// TIA Portal V16 export
// export: Created 2022-11-17T15:49:30.6302433Z, ExportSetting WithDefaults, DisplayName Totally Integrated Automation Portal, DisplayVersion V16 Update 6, DisplayName TIA Portal Version Control Interface, DisplayVersion V16 Update 2, DisplayName TIA Portal Openness, DisplayVersion V16 Update 6, DisplayName SINAMICS Startdrive Advanced, DisplayVersion V16 Update 5, DisplayName SINAMICS Startdrive G130, G150, S120, S150, SINAMICS MV, S210, DisplayVersion V16 Update 5, DisplayName SINAMICS Startdrive G110M, G120, G120C, G120D, G120P, G115D, DisplayVersion V16 Update 5, DisplayName STEP 7 Professional, DisplayVersion V16 Update 6, DisplayName STEP 7 Safety, DisplayVersion V16, DisplayName WinCC Advanced, DisplayVersion V16 Update 6
FUNCTION "FC90_PageManagement" : Void   // FC90, LAD
{ S7_Optimized_Access := 'FALSE' }
VERSION : 0.1
// stored: AutoNumber false, IsIECCheckEnabled false, SetENOAutomatically false, UDAEnableTagReadback false
   VAR_TEMP
      CurrentPage : Int;
      PageBkwRequest : Int;
      PageFwRequest : Int;
   END_VAR
   VAR_TEMP   // added for the SCL form of the ladder/FBD networks
      _w1 : Bool;
   END_VAR
BEGIN

REGION Network 1
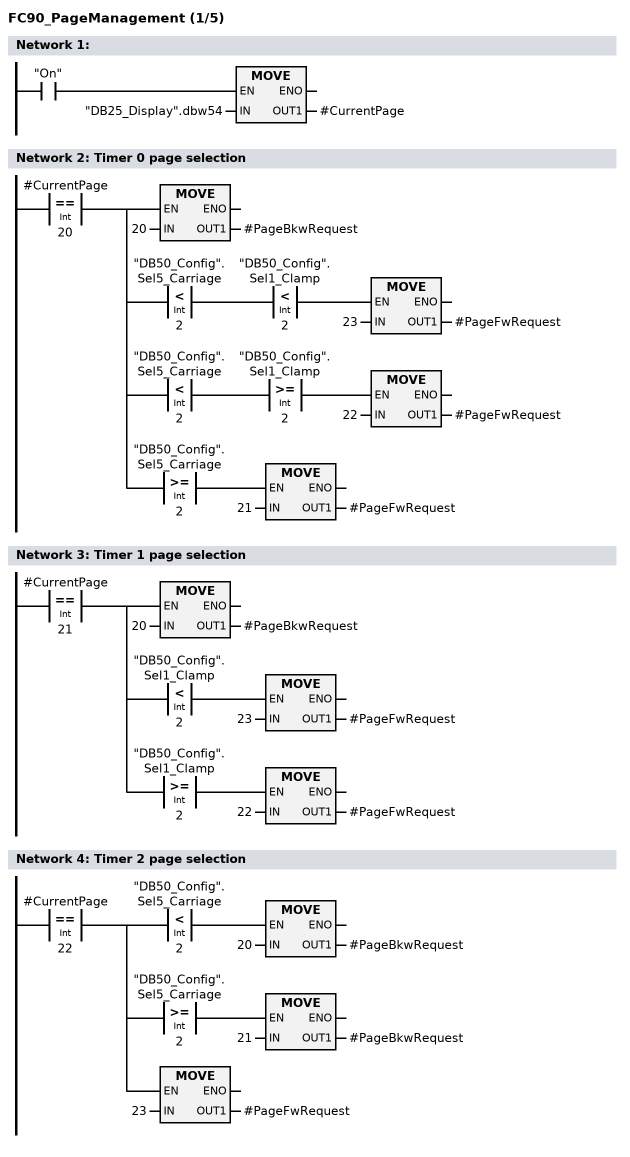
   RUNG wire#powerrail
      Contact( "On" )
      { S7_GenerateENO := "TRUE" } Move(in := "DB25_Display".dbw54, out1 => #CurrentPage)
   END_RUNG
   // the same network as SCL:
   IF "On" THEN #CurrentPage := "DB25_Display".dbw54; END_IF;
END_REGION

REGION Network 2: Timer 0 page selection
   RUNG wire#powerrail
      { S7_Templates := "SrcType := Int" } EQ_Contact(in1 := #CurrentPage, in2 := 20)
      wire#w1
      { S7_GenerateENO := "TRUE" } Move(in := 20, out1 => #PageBkwRequest)
   END_RUNG
   RUNG wire#w1
      { S7_Templates := "SrcType := Int" } LT_Contact(in1 := "DB50_Config".Sel5_Carriage, in2 := 2)
      { S7_Templates := "SrcType := Int" } LT_Contact(in1 := "DB50_Config".Sel1_Clamp, in2 := 2)
      { S7_GenerateENO := "TRUE" } Move(in := 23, out1 => #PageFwRequest)
   END_RUNG
   RUNG wire#w1
      { S7_Templates := "SrcType := Int" } LT_Contact(in1 := "DB50_Config".Sel5_Carriage, in2 := 2)
      { S7_Templates := "SrcType := Int" } GE_Contact(in1 := "DB50_Config".Sel1_Clamp, in2 := 2)
      { S7_GenerateENO := "TRUE" } Move(in := 22, out1 => #PageFwRequest)
   END_RUNG
   RUNG wire#w1
      { S7_Templates := "SrcType := Int" } GE_Contact(in1 := "DB50_Config".Sel5_Carriage, in2 := 2)
      { S7_GenerateENO := "TRUE" } Move(in := 21, out1 => #PageFwRequest)
   END_RUNG
   // the same network as SCL:
   #_w1 := #CurrentPage = 20;
   IF #_w1 THEN #PageBkwRequest := 20; END_IF;
   IF #_w1 AND ("DB50_Config".Sel5_Carriage < 2) AND ("DB50_Config".Sel1_Clamp < 2) THEN
       #PageFwRequest := 23;
   END_IF;
   IF #_w1 AND ("DB50_Config".Sel5_Carriage < 2) AND ("DB50_Config".Sel1_Clamp >= 2) THEN
       #PageFwRequest := 22;
   END_IF;
   IF #_w1 AND ("DB50_Config".Sel5_Carriage >= 2) THEN #PageFwRequest := 21; END_IF;
END_REGION

REGION Network 3: Timer 1 page selection
   RUNG wire#powerrail
      { S7_Templates := "SrcType := Int" } EQ_Contact(in1 := #CurrentPage, in2 := 21)
      wire#w1
      { S7_GenerateENO := "TRUE" } Move(in := 20, out1 => #PageBkwRequest)
   END_RUNG
   RUNG wire#w1
      { S7_Templates := "SrcType := Int" } LT_Contact(in1 := "DB50_Config".Sel1_Clamp, in2 := 2)
      { S7_GenerateENO := "TRUE" } Move(in := 23, out1 => #PageFwRequest)
   END_RUNG
   RUNG wire#w1
      { S7_Templates := "SrcType := Int" } GE_Contact(in1 := "DB50_Config".Sel1_Clamp, in2 := 2)
      { S7_GenerateENO := "TRUE" } Move(in := 22, out1 => #PageFwRequest)
   END_RUNG
   // the same network as SCL:
   #_w1 := #CurrentPage = 21;
   IF #_w1 THEN #PageBkwRequest := 20; END_IF;
   IF #_w1 AND ("DB50_Config".Sel1_Clamp < 2) THEN #PageFwRequest := 23; END_IF;
   IF #_w1 AND ("DB50_Config".Sel1_Clamp >= 2) THEN #PageFwRequest := 22; END_IF;
END_REGION

REGION Network 4: Timer 2 page selection
   RUNG wire#powerrail
      { S7_Templates := "SrcType := Int" } EQ_Contact(in1 := #CurrentPage, in2 := 22)
      wire#w1
      { S7_Templates := "SrcType := Int" } LT_Contact(in1 := "DB50_Config".Sel5_Carriage, in2 := 2)
      { S7_GenerateENO := "TRUE" } Move(in := 20, out1 => #PageBkwRequest)
   END_RUNG
   RUNG wire#w1
      { S7_Templates := "SrcType := Int" } GE_Contact(in1 := "DB50_Config".Sel5_Carriage, in2 := 2)
      { S7_GenerateENO := "TRUE" } Move(in := 21, out1 => #PageBkwRequest)
   END_RUNG
   RUNG wire#w1
      { S7_GenerateENO := "TRUE" } Move(in := 23, out1 => #PageFwRequest)
   END_RUNG
   // the same network as SCL:
   #_w1 := #CurrentPage = 22;
   IF #_w1 AND ("DB50_Config".Sel5_Carriage < 2) THEN #PageBkwRequest := 20; END_IF;
   IF #_w1 AND ("DB50_Config".Sel5_Carriage >= 2) THEN #PageBkwRequest := 21; END_IF;
   IF #_w1 THEN #PageFwRequest := 23; END_IF;
END_REGION

REGION Network 5: Timer 3 page selection
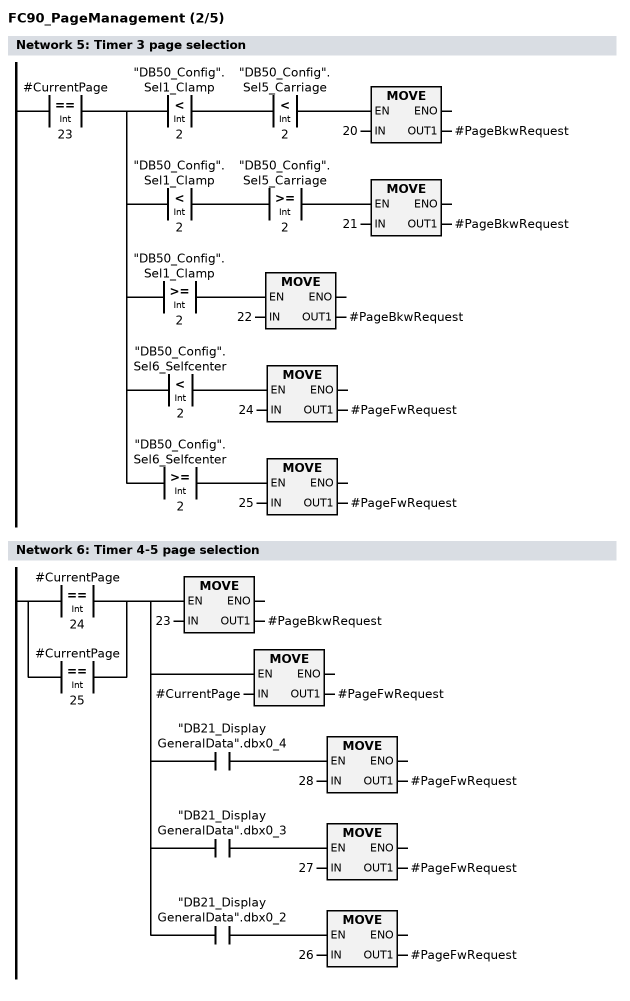
   RUNG wire#powerrail
      { S7_Templates := "SrcType := Int" } EQ_Contact(in1 := #CurrentPage, in2 := 23)
      wire#w1
      { S7_Templates := "SrcType := Int" } LT_Contact(in1 := "DB50_Config".Sel1_Clamp, in2 := 2)
      { S7_Templates := "SrcType := Int" } LT_Contact(in1 := "DB50_Config".Sel5_Carriage, in2 := 2)
      { S7_GenerateENO := "TRUE" } Move(in := 20, out1 => #PageBkwRequest)
   END_RUNG
   RUNG wire#w1
      { S7_Templates := "SrcType := Int" } LT_Contact(in1 := "DB50_Config".Sel1_Clamp, in2 := 2)
      { S7_Templates := "SrcType := Int" } GE_Contact(in1 := "DB50_Config".Sel5_Carriage, in2 := 2)
      { S7_GenerateENO := "TRUE" } Move(in := 21, out1 => #PageBkwRequest)
   END_RUNG
   RUNG wire#w1
      { S7_Templates := "SrcType := Int" } GE_Contact(in1 := "DB50_Config".Sel1_Clamp, in2 := 2)
      { S7_GenerateENO := "TRUE" } Move(in := 22, out1 => #PageBkwRequest)
   END_RUNG
   RUNG wire#w1
      { S7_Templates := "SrcType := Int" } LT_Contact(in1 := "DB50_Config".Sel6_Selfcenter, in2 := 2)
      { S7_GenerateENO := "TRUE" } Move(in := 24, out1 => #PageFwRequest)
   END_RUNG
   RUNG wire#w1
      { S7_Templates := "SrcType := Int" } GE_Contact(in1 := "DB50_Config".Sel6_Selfcenter, in2 := 2)
      { S7_GenerateENO := "TRUE" } Move(in := 25, out1 => #PageFwRequest)
   END_RUNG
   // the same network as SCL:
   #_w1 := #CurrentPage = 23;
   IF #_w1 AND ("DB50_Config".Sel1_Clamp < 2) AND ("DB50_Config".Sel5_Carriage < 2) THEN
       #PageBkwRequest := 20;
   END_IF;
   IF #_w1 AND ("DB50_Config".Sel1_Clamp < 2) AND ("DB50_Config".Sel5_Carriage >= 2) THEN
       #PageBkwRequest := 21;
   END_IF;
   IF #_w1 AND ("DB50_Config".Sel1_Clamp >= 2) THEN #PageBkwRequest := 22; END_IF;
   IF #_w1 AND ("DB50_Config".Sel6_Selfcenter < 2) THEN #PageFwRequest := 24; END_IF;
   IF #_w1 AND ("DB50_Config".Sel6_Selfcenter >= 2) THEN #PageFwRequest := 25; END_IF;
END_REGION

REGION Network 6: Timer 4-5 page selection
   RUNG wire#powerrail
      { S7_Templates := "SrcType := Int" } EQ_Contact(in1 := #CurrentPage, in2 := 24)
      wire#w1
      { S7_GenerateENO := "TRUE" } Move(in := 23, out1 => #PageBkwRequest)
   END_RUNG
   RUNG wire#powerrail
      { S7_Templates := "SrcType := Int" } EQ_Contact(in1 := #CurrentPage, in2 := 25)
   END_RUNG wire#w1
   RUNG wire#w1
      { S7_GenerateENO := "TRUE" } Move(in := #CurrentPage, out1 => #PageFwRequest)
   END_RUNG
   RUNG wire#w1
      Contact( "DB21_DisplayGeneralData".dbx0_4 )
      { S7_GenerateENO := "TRUE" } Move(in := 28, out1 => #PageFwRequest)
   END_RUNG
   RUNG wire#w1
      Contact( "DB21_DisplayGeneralData".dbx0_3 )
      { S7_GenerateENO := "TRUE" } Move(in := 27, out1 => #PageFwRequest)
   END_RUNG
   RUNG wire#w1
      Contact( "DB21_DisplayGeneralData".dbx0_2 )
      { S7_GenerateENO := "TRUE" } Move(in := 26, out1 => #PageFwRequest)
   END_RUNG
   // the same network as SCL:
   #_w1 := (#CurrentPage = 24) OR (#CurrentPage = 25);
   IF #_w1 THEN
       #PageBkwRequest := 23;
       #PageFwRequest := #CurrentPage;
   END_IF;
   IF #_w1 AND "DB21_DisplayGeneralData".dbx0_4 THEN #PageFwRequest := 28; END_IF;
   IF #_w1 AND "DB21_DisplayGeneralData".dbx0_3 THEN #PageFwRequest := 27; END_IF;
   IF #_w1 AND "DB21_DisplayGeneralData".dbx0_2 THEN #PageFwRequest := 26; END_IF;
END_REGION

REGION Network 7: Timer 6 page selection
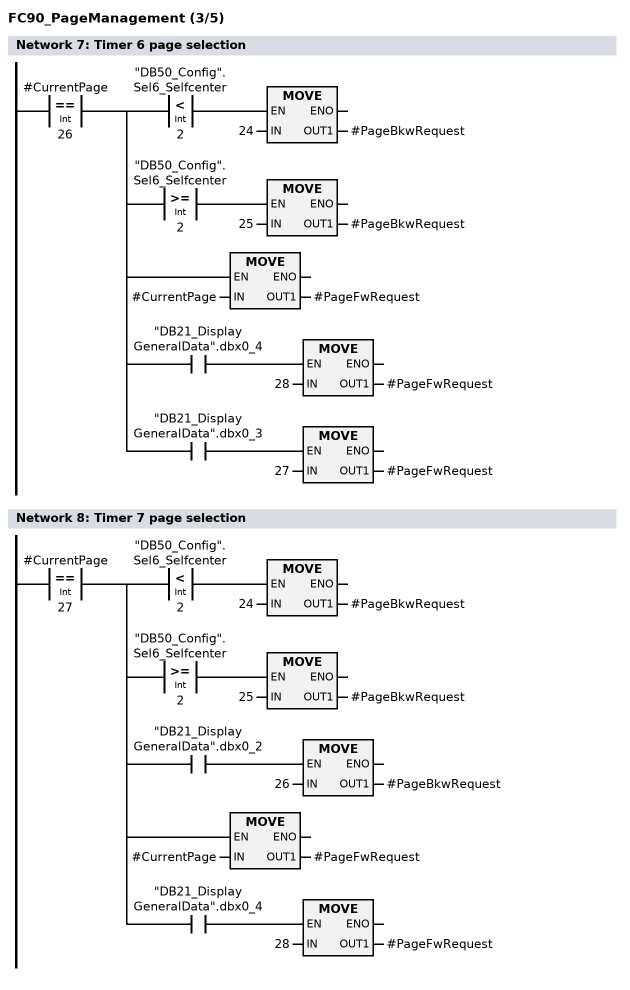
   RUNG wire#powerrail
      { S7_Templates := "SrcType := Int" } EQ_Contact(in1 := #CurrentPage, in2 := 26)
      wire#w1
      { S7_Templates := "SrcType := Int" } LT_Contact(in1 := "DB50_Config".Sel6_Selfcenter, in2 := 2)
      { S7_GenerateENO := "TRUE" } Move(in := 24, out1 => #PageBkwRequest)
   END_RUNG
   RUNG wire#w1
      { S7_Templates := "SrcType := Int" } GE_Contact(in1 := "DB50_Config".Sel6_Selfcenter, in2 := 2)
      { S7_GenerateENO := "TRUE" } Move(in := 25, out1 => #PageBkwRequest)
   END_RUNG
   RUNG wire#w1
      { S7_GenerateENO := "TRUE" } Move(in := #CurrentPage, out1 => #PageFwRequest)
   END_RUNG
   RUNG wire#w1
      Contact( "DB21_DisplayGeneralData".dbx0_4 )
      { S7_GenerateENO := "TRUE" } Move(in := 28, out1 => #PageFwRequest)
   END_RUNG
   RUNG wire#w1
      Contact( "DB21_DisplayGeneralData".dbx0_3 )
      { S7_GenerateENO := "TRUE" } Move(in := 27, out1 => #PageFwRequest)
   END_RUNG
   // the same network as SCL:
   #_w1 := #CurrentPage = 26;
   IF #_w1 AND ("DB50_Config".Sel6_Selfcenter < 2) THEN #PageBkwRequest := 24; END_IF;
   IF #_w1 AND ("DB50_Config".Sel6_Selfcenter >= 2) THEN #PageBkwRequest := 25; END_IF;
   IF #_w1 THEN #PageFwRequest := #CurrentPage; END_IF;
   IF #_w1 AND "DB21_DisplayGeneralData".dbx0_4 THEN #PageFwRequest := 28; END_IF;
   IF #_w1 AND "DB21_DisplayGeneralData".dbx0_3 THEN #PageFwRequest := 27; END_IF;
END_REGION

REGION Network 8: Timer 7 page selection
   RUNG wire#powerrail
      { S7_Templates := "SrcType := Int" } EQ_Contact(in1 := #CurrentPage, in2 := 27)
      wire#w1
      { S7_Templates := "SrcType := Int" } LT_Contact(in1 := "DB50_Config".Sel6_Selfcenter, in2 := 2)
      { S7_GenerateENO := "TRUE" } Move(in := 24, out1 => #PageBkwRequest)
   END_RUNG
   RUNG wire#w1
      { S7_Templates := "SrcType := Int" } GE_Contact(in1 := "DB50_Config".Sel6_Selfcenter, in2 := 2)
      { S7_GenerateENO := "TRUE" } Move(in := 25, out1 => #PageBkwRequest)
   END_RUNG
   RUNG wire#w1
      Contact( "DB21_DisplayGeneralData".dbx0_2 )
      { S7_GenerateENO := "TRUE" } Move(in := 26, out1 => #PageBkwRequest)
   END_RUNG
   RUNG wire#w1
      { S7_GenerateENO := "TRUE" } Move(in := #CurrentPage, out1 => #PageFwRequest)
   END_RUNG
   RUNG wire#w1
      Contact( "DB21_DisplayGeneralData".dbx0_4 )
      { S7_GenerateENO := "TRUE" } Move(in := 28, out1 => #PageFwRequest)
   END_RUNG
   // the same network as SCL:
   #_w1 := #CurrentPage = 27;
   IF #_w1 AND ("DB50_Config".Sel6_Selfcenter < 2) THEN #PageBkwRequest := 24; END_IF;
   IF #_w1 AND ("DB50_Config".Sel6_Selfcenter >= 2) THEN #PageBkwRequest := 25; END_IF;
   IF #_w1 AND "DB21_DisplayGeneralData".dbx0_2 THEN #PageBkwRequest := 26; END_IF;
   IF #_w1 THEN #PageFwRequest := #CurrentPage; END_IF;
   IF #_w1 AND "DB21_DisplayGeneralData".dbx0_4 THEN #PageFwRequest := 28; END_IF;
END_REGION

REGION Network 9: Timer 8 page selection
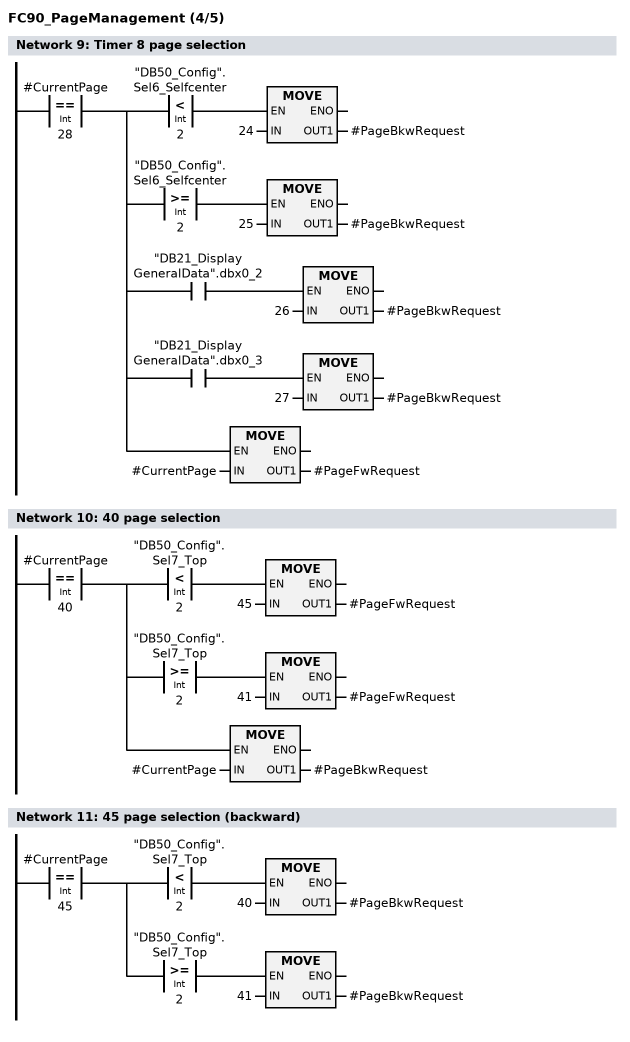
   RUNG wire#powerrail
      { S7_Templates := "SrcType := Int" } EQ_Contact(in1 := #CurrentPage, in2 := 28)
      wire#w1
      { S7_Templates := "SrcType := Int" } LT_Contact(in1 := "DB50_Config".Sel6_Selfcenter, in2 := 2)
      { S7_GenerateENO := "TRUE" } Move(in := 24, out1 => #PageBkwRequest)
   END_RUNG
   RUNG wire#w1
      { S7_Templates := "SrcType := Int" } GE_Contact(in1 := "DB50_Config".Sel6_Selfcenter, in2 := 2)
      { S7_GenerateENO := "TRUE" } Move(in := 25, out1 => #PageBkwRequest)
   END_RUNG
   RUNG wire#w1
      Contact( "DB21_DisplayGeneralData".dbx0_2 )
      { S7_GenerateENO := "TRUE" } Move(in := 26, out1 => #PageBkwRequest)
   END_RUNG
   RUNG wire#w1
      Contact( "DB21_DisplayGeneralData".dbx0_3 )
      { S7_GenerateENO := "TRUE" } Move(in := 27, out1 => #PageBkwRequest)
   END_RUNG
   RUNG wire#w1
      { S7_GenerateENO := "TRUE" } Move(in := #CurrentPage, out1 => #PageFwRequest)
   END_RUNG
   // the same network as SCL:
   #_w1 := #CurrentPage = 28;
   IF #_w1 AND ("DB50_Config".Sel6_Selfcenter < 2) THEN #PageBkwRequest := 24; END_IF;
   IF #_w1 AND ("DB50_Config".Sel6_Selfcenter >= 2) THEN #PageBkwRequest := 25; END_IF;
   IF #_w1 AND "DB21_DisplayGeneralData".dbx0_2 THEN #PageBkwRequest := 26; END_IF;
   IF #_w1 AND "DB21_DisplayGeneralData".dbx0_3 THEN #PageBkwRequest := 27; END_IF;
   IF #_w1 THEN #PageFwRequest := #CurrentPage; END_IF;
END_REGION

REGION Network 10: 40 page selection
   RUNG wire#powerrail
      { S7_Templates := "SrcType := Int" } EQ_Contact(in1 := #CurrentPage, in2 := 40)
      wire#w1
      { S7_Templates := "SrcType := Int" } LT_Contact(in1 := "DB50_Config".Sel7_Top, in2 := 2)
      { S7_GenerateENO := "TRUE" } Move(in := 45, out1 => #PageFwRequest)
   END_RUNG
   RUNG wire#w1
      { S7_Templates := "SrcType := Int" } GE_Contact(in1 := "DB50_Config".Sel7_Top, in2 := 2)
      { S7_GenerateENO := "TRUE" } Move(in := 41, out1 => #PageFwRequest)
   END_RUNG
   RUNG wire#w1
      { S7_GenerateENO := "TRUE" } Move(in := #CurrentPage, out1 => #PageBkwRequest)
   END_RUNG
   // the same network as SCL:
   #_w1 := #CurrentPage = 40;
   IF #_w1 AND ("DB50_Config".Sel7_Top < 2) THEN #PageFwRequest := 45; END_IF;
   IF #_w1 AND ("DB50_Config".Sel7_Top >= 2) THEN #PageFwRequest := 41; END_IF;
   IF #_w1 THEN #PageBkwRequest := #CurrentPage; END_IF;
END_REGION

REGION Network 11: 45 page selection (backward)
   RUNG wire#powerrail
      { S7_Templates := "SrcType := Int" } EQ_Contact(in1 := #CurrentPage, in2 := 45)
      wire#w1
      { S7_Templates := "SrcType := Int" } LT_Contact(in1 := "DB50_Config".Sel7_Top, in2 := 2)
      { S7_GenerateENO := "TRUE" } Move(in := 40, out1 => #PageBkwRequest)
   END_RUNG
   RUNG wire#w1
      { S7_Templates := "SrcType := Int" } GE_Contact(in1 := "DB50_Config".Sel7_Top, in2 := 2)
      { S7_GenerateENO := "TRUE" } Move(in := 41, out1 => #PageBkwRequest)
   END_RUNG
   // the same network as SCL:
   #_w1 := #CurrentPage = 45;
   IF #_w1 AND ("DB50_Config".Sel7_Top < 2) THEN #PageBkwRequest := 40; END_IF;
   IF #_w1 AND ("DB50_Config".Sel7_Top >= 2) THEN #PageBkwRequest := 41; END_IF;
END_REGION

REGION Network 12
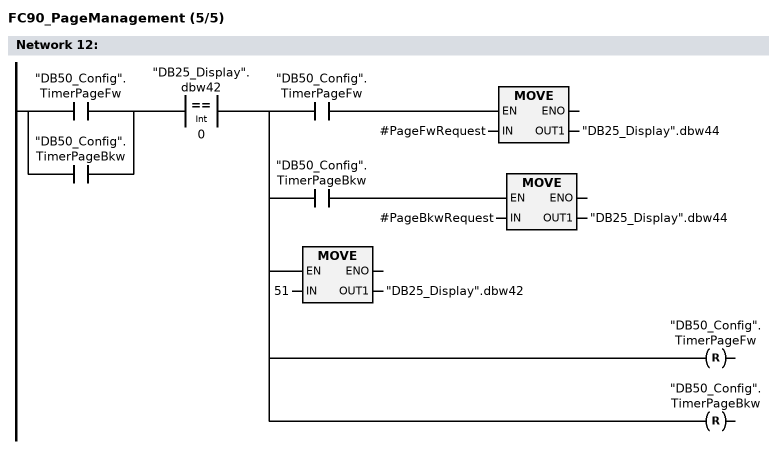
   RUNG wire#powerrail
      Contact( "DB50_Config".TimerPageFw )
      wire#w1
      { S7_Templates := "SrcType := Int" } EQ_Contact(in1 := "DB25_Display".dbw42, in2 := 0)
      wire#w2
      Contact( "DB50_Config".TimerPageFw )
      { S7_GenerateENO := "TRUE" } Move(in := #PageFwRequest, out1 => "DB25_Display".dbw44)
   END_RUNG
   RUNG wire#powerrail
      Contact( "DB50_Config".TimerPageBkw )
   END_RUNG wire#w1
   RUNG wire#w2
      Contact( "DB50_Config".TimerPageBkw )
      { S7_GenerateENO := "TRUE" } Move(in := #PageBkwRequest, out1 => "DB25_Display".dbw44)
   END_RUNG
   RUNG wire#w2
      { S7_GenerateENO := "TRUE" } Move(in := 51, out1 => "DB25_Display".dbw42)
   END_RUNG
   RUNG wire#w2
      R_Coil( "DB50_Config".TimerPageFw )
   END_RUNG
   RUNG wire#w2
      R_Coil( "DB50_Config".TimerPageBkw )
   END_RUNG
   // the same network as SCL:
   #_w1 := ("DB50_Config".TimerPageFw OR "DB50_Config".TimerPageBkw) AND ("DB25_Display".dbw42 = 0);
   IF #_w1 AND "DB50_Config".TimerPageFw THEN "DB25_Display".dbw44 := #PageFwRequest; END_IF;
   IF #_w1 AND "DB50_Config".TimerPageBkw THEN "DB25_Display".dbw44 := #PageBkwRequest; END_IF;
   IF #_w1 THEN
       "DB25_Display".dbw42 := 51;
       "DB50_Config".TimerPageFw := FALSE;
       "DB50_Config".TimerPageBkw := FALSE;
   END_IF;
END_REGION
END_FUNCTION
